FUNCTION FUN_In_Zone : BOOL
VAR_INPUT
	Current  : LREAL;
	Required : LREAL;
	Margin    : LREAL;
END_VAR
VAR
END_VAR

IF ((Current) < (Required + Margin )) AND ((Current) > (Required - Margin)) THEN
	FUN_In_Zone := TRUE;
ELSE
	FUN_In_Zone := FALSE;
END_IF

END_FUNCTION

(* stored: Version 1.1.0.1, ProductVersion 3.1.4024.4
   POU FUN_In_Zone: Id {ee824f19-0c97-4ccf-95e1-b33b83f62b4e}, SpecialFunc None *)
